FUNCTION_BLOCK TcGraph IMPLEMENTS I_TcGraph
VAR
	nodeFactories : NodeFactorys;
	linkFactory : LinkFactory;
END_VAR

METHOD PUBLIC Accept
VAR_INPUT
	Visitor : I_TcGraphVisitor;
END_VAR
Visitor.VisitTcGraph(this^);
END_METHOD

METHOD PUBLIC GetNodeFactories : I_NodeFactorys
VAR_INPUT
END_VAR
GetNodeFactories := nodeFactories;
END_METHOD

METHOD PUBLIC InstallNodePack
VAR_INPUT
	NodePack : I_NodePack;
END_VAR
NodePack.RegisterWithGraph(This^);
END_METHOD

METHOD PUBLIC NewGraph : I_Graph
VAR_INPUT
END_VAR
VAR
	pGraph : POINTER TO Graph;
END_VAR
pGraph := __NEW(Graph(NodeFactories:= THIS^.nodeFactories,LinkFactory := THIS^.linkFactory));
NewGraph := pGraph^;
END_METHOD

METHOD PUBLIC RegisterNodeFactoryByType
VAR_INPUT
	NodeType : T_MAXSTRING;
	NodeFactory : I_NodeFactory;	
END_VAR
nodeFactories.InsertByType(NodeType,NodeFactory);
{warning <'should add event here'>}
END_METHOD

END_FUNCTION_BLOCK

(* stored: Version 1.1.0.1, ProductVersion 3.1.4024.12
   POU TcGraph: Id {3cf4dffb-2e67-0cde-05c3-0b7a44e6e216}, SpecialFunc None
   Method Accept: Id {d8350354-5d0e-015a-02f7-c388e7f54195}
   Method GetNodeFactories: Id {c44bbbb1-a7c9-06c4-05cd-ffa320ca8ae8}
   Method InstallNodePack: Id {0ec00c43-b35f-0669-2893-bc57927b1baa}
   Method NewGraph: Id {3dacf3c5-2186-0d1e-08e0-d29f6557f3d4}
   Method RegisterNodeFactoryByType: Id {e69125b8-4a8c-01f5-3b08-4f76913c652b} *)
